            // --- Phase 1: ToolHeadLock verification ------------------------------------
            // Cmd_Extend is held TRUE for the whole of PAUSED (see the ToolHeadLock section
            // at the bottom of this FB), so the lock is already COMMANDED in the entire time
            // the machine sits paused. This phase adds the WAIT, not the command.
            //
            // Why it is needed: PAUSED used to go straight to RUNNING, so nothing re-checked
            // the lock on resume. FC_CylinderDispatch is not gated on machine state, so an
            // operator can retract the lock from the manual cylinder page while paused — in
            // cylinder FB State 3 the Cmd_Retract/Cmd_RetractFull test comes BEFORE the
            // process's Cmd_Extend, so the HMI button wins. It also catches a purely
            // mechanical failure to re-engage, which no HMI-side gate would ever see.
            //
            // Same three-way test and same error code as STATE_LOCK_EXTEND_WAIT (17), so the
            // two lock-confirm paths cannot drift apart. It cannot hang: Cmd_Extend is
            // asserted throughout, so the cylinder FB reaches either AtSetpoint or its own
            // Timeout_Extend → Error. Error_Text/ErrorDetail name the resume path so the
            // online trail still distinguishes this from a state-17 failure.
            IF #bResumeLockChk THEN
                IF "DB_HMI".Bypass_ToolHeadLock OR "DB_Cylinder_ToolHeadLock".AtSetpoint THEN
                    #bResumeLockChk := FALSE;
                    #bResumeSpeedup := TRUE;      // lock confirmed → start the spindle spin-up
                ELSIF "DB_Cylinder_ToolHeadLock".Error THEN
                    #bResumeLockChk := FALSE;
                    #newErrorFlag := TRUE;
                    #newErrorCode := 16#0012;
                    "DB_Diagnostic".Error_Text := 'PauseResume: ToolHeadLock not engaged - CylFB.Error=TRUE, AtSetpoint=FALSE';
                    "DB_HMI".ErrorDetail    := 'Tool head lock not engaged on resume - check cylinder/sensor';
                    #State := STATE_ERROR;
                END_IF;
            END_IF;

            // --- Phase 2: spindle spin-up ----------------------------------------------
            IF #bResumeSpeedup AND #tonResumeSpeedup.Q THEN
                #bResumeSpeedup := FALSE;
                #bPauseActive   := FALSE;
                #State          := STATE_RUNNING;
            END_IF;

        // -----------------------------------------------------------------
        // === STATE_TOOL_CHANGE (30) ===
        // -----------------------------------------------------------------
        30: // TOOL_CHANGE
            #StatusID := 4; #bToolExecute := TRUE; #State := STATE_TOOL_WAIT;

        // -----------------------------------------------------------------
        // === STATE_TOOL_WAIT (35) ===
        // -----------------------------------------------------------------
        35: // TOOL_WAIT
            IF #fbToolChanger.Done THEN
                #bToolExecute := FALSE;
                #CurrentTool := #fbToolChanger.CurrentTool;
                #fbRecipeHandler.ToolChangeReq := FALSE;  // Signal RecipeHandler to continue
                // Tool change done: re-engage lock before resuming machining
                #State := STATE_LOCK_EXTEND_WAIT;
            ELSIF #fbToolChanger.Error THEN
                #bToolExecute := FALSE;
                #State := STATE_ERROR;
                #newErrorFlag := TRUE;
                #newErrorCode := #fbToolChanger.ErrorID;
                "DB_HMI".ErrorDetail    := CONCAT(IN1 := 'Tool ', IN2 := INT_TO_STRING(#activeToolReq));
            END_IF;

        // -----------------------------------------------------------------
        // === STATE_ERROR (999) ===
        // -----------------------------------------------------------------
        999: // ERROR
            #StatusID := 99; #bStartSeq := FALSE; #Error := TRUE;
            #bRecipeLoadExec := FALSE;   // a recipe copy must not stay in flight across an error ack
            #timerRunning := FALSE;  // Stop cycle timer
            #bResumeSpeedup := FALSE;  // Cancel any pending pause spin-up wait (e.g. fault during spin-up)
            #bResumeLockChk := FALSE;  // Cancel any pending pause lock verification
            // Cancel any pending STOPPING spindle-decel wait. Added with ITEM-56c, but it also
            // closes a route that already existed: STATE_STOPPING could be left for STATE_ERROR by
            // an E-Stop or safety fault, and NOTHING cleared this flag on that path (only phase 2
            // itself and the hard reset did). A stale TRUE makes the NEXT stop skip phase 1
            // entirely -- no spindle stop command, no park move, no sheet-holder release -- and
            // drop straight into phase 2 on a leftover spindleStopPT. Level-cleared here every
            // scan while faulted, so no acknowledge path can miss it.
            #bWaitingSpindleStop := FALSE;
            // Cancel the end-of-program sanding dwell (2026-08-29) and drop the spindle
            // command it raised. A safety fault (E-Stop, air) during the dwell forces
            // STATE_ERROR from COMPLETE via the safety block above, and bDrivesEnable
            // already stops the spindle -- but STATE_COMPLETE is the only block that
            // clears #bSpindleStart on this path, and it no longer runs once State is 999.
            // Level-cleared every scan while faulted, so no acknowledge path can miss it.
            #bSandActive   := FALSE;
            #bSpindleStart := FALSE;
            // Clear the BackSupport atmosphere valve — de-energises on error.
            // Cmd_Retract is deliberately NOT touched here: the end-of-recipe retract
            // block (bottom of this FB) owns it and needs it held for the retract window.
            "DB_Cylinder_BackSupport".SolAtmo_Cmd := FALSE;
            // Clear BackSupport extend (recipe CMD=40 or manual button/MDI) while faulted
            "DB_Cylinder_BackSupport".Cmd_Extend  := FALSE;
            #bMDI_Cmd40Extend                     := FALSE;
            // CMD=41 edge memory: seed with the live button state while faulted, so a
            // button held through the fault cannot fire a one-shot after acknowledge.
            #prevBtnCmd41Release := "DB_Manual".Btn_Cmd41_Release;
            #prevBtnCmd41AtmoOff := "DB_Manual".Btn_Cmd41_AtmoOff;
            #prevBtnCmd41AtmoOn  := "DB_Manual".Btn_Cmd41_AtmoOn;
            // SheetHolder Cmd_Extend is driven FALSE here by its single writer at the bottom of
            // this FB (State <> SHEET_WAIT), so it cannot hold through an error acknowledge.

            // Save current position for warm restart
            IF #savedLineIndex < 0 THEN
                #savedLineIndex := #fbRecipeHandler.CurrentLine;
                #savedProgram := #activeProgram;
            END_IF;
            "DB_HMI".ResumeLine := #savedLineIndex;   // HMI shows which line will be resumed on next Start

            // Debug: populate DB_Diagnostic with error context for easier troubleshooting
            // Error_ProcessState is deliberately NOT written here: this block only runs in
            // STATE_ERROR, so it could only ever record 999. It is captured at alarm time
            // instead -- see the guarded write before the FB_AlarmManager call.
            "DB_Diagnostic".Error_Code := #fbAlarmManager.ActiveErrorCode; // primary error source
            // If recipe handler provided an error line, prefer that
            IF "DB_Diagnostic".Recipe_CurrentLine >= 0 THEN
                "DB_Diagnostic".Error_Line := "DB_Diagnostic".Recipe_CurrentLine;
            END_IF;

            // BUG FIX: Previous implementation transitioned ackEdge → STATE_PAUSED,
            // but the recipe handler remained in its internal STATE_ERROR (999).
            // In PAUSED → Continue → STATE_RUNNING the recipe handler was not running (error state).
            // Fix: All recovery paths go to STATE_STOPPED + recipe handler is reset.
            // When operator presses Start, PRE_SCAN → STARTING → RUNNING flow starts clean.
            // ACK, Continue and Restart are blocked while E-Stop is active.
            // E-Stop must be physically released before any error acknowledgement is accepted.
            IF #ackEdge AND (#EStop_OK OR "DB_HMI".Bypass_EStop) THEN
                // Acknowledge: clear error → STOPPED. savedLineIndex kept for warm restart on next Start.
                #Error := FALSE;
                #bPauseActive := FALSE;
                #bResetRecipe := TRUE;   // Reset recipe handler to IDLE (cannot continue from state 999)
                #prevSafetyError := FALSE;   // Clear safety latch -- fresh evaluation on restart
                #bSheetWaitPhase2         := FALSE;
                #bSheetWaitPhase3         := FALSE;
                IF NOT "DB_MachineConfig".Bypass_MandrelLock THEN
                    #bMandrelRetractPending := TRUE;  // ITEM-32: deferred — spindle may still be spinning; wait SpindleStopSafeTime
                END_IF;
                #bSheetHolderRetractHold  := TRUE;  // Release sheet holder (may be extended from last run)
                #fbAlarmManager(NewError := FALSE, NewErrorCode := 0,
                                AcknowledgeError := TRUE);
                #State := STATE_STOPPED;
            ELSIF #continueEdge AND (#EStop_OK OR "DB_HMI".Bypass_EStop) THEN
                // Continue: resume from savedLineIndex on next Start (warm restart)
                #Error := FALSE;
                #bPauseActive := FALSE;
                #bResetRecipe := TRUE;
                #bSheetWaitPhase2         := FALSE;
                #bSheetWaitPhase3         := FALSE;
                IF NOT "DB_MachineConfig".Bypass_MandrelLock THEN
                    #bMandrelRetractPending := TRUE;  // ITEM-32: deferred — spindle may still be spinning; wait SpindleStopSafeTime
                END_IF;
                #bSheetHolderRetractHold  := TRUE;  // Release sheet holder
                #fbAlarmManager(NewError := FALSE, NewErrorCode := 0,
                                AcknowledgeError := TRUE);
                #State := STATE_STOPPED;
            ELSIF #restartEdge AND (#EStop_OK OR "DB_HMI".Bypass_EStop) THEN
                // Restart: explicit restart from line 0 -- clear saved position
                #Error := FALSE;
                #bPauseActive := FALSE;
                #bResetRecipe := TRUE;
                #savedLineIndex := -1;
                #savedProgram := -1;
                "DB_HMI".ResumeLine := -1;
                #bSheetWaitPhase2         := FALSE;
                #bSheetWaitPhase3         := FALSE;
                IF NOT "DB_MachineConfig".Bypass_MandrelLock THEN
                    #bMandrelRetractPending := TRUE;  // ITEM-32: deferred — spindle may still be spinning; wait SpindleStopSafeTime
                END_IF;
                #bSheetHolderRetractHold  := TRUE;  // Release sheet holder
                #fbAlarmManager(NewError := FALSE, NewErrorCode := 0,
                                AcknowledgeError := TRUE);
                #State := STATE_STOPPED;
            END_IF;
    END_CASE;

    // -----------------------------------------------------------------
    // === STATE_COMPLETE (100) ===
    // (handled as IF block outside CASE -- no new constant needed)
    // -----------------------------------------------------------------
    IF #State = 100 THEN
        #StatusID := 100; #bStartSeq := FALSE;
        #Running := FALSE;
        // Clear bSpindleStart: RUNNING no longer runs to clear it, so SpindleReqStart=TRUE
        // from the last CMD_SPINDLE_ON would keep Start=TRUE through PRE_SCAN and STARTING.
        // prevStart is reset inside FB_SpindleControl on halt Done, so the next CMD_SPINDLE_ON
        // in the new recipe generates a clean startEdge.
        // bSpindleStop is intentionally NOT cleared here. (The old comment claimed the Done
        // handler in CASE 20 sets it, and that clearing it in the same scan would cancel the
        // stop. That was already wrong before this change and is corrected 2026-08-29:
        // #bSpindleStop is set in exactly ONE place, STATE_STOPPING phase 1 -- the completion
        // path never raises it. It is cleared in STATE_STOPPED. Nothing to do here either way.)
        //
        // SANDING DWELL (2026-08-29): the one exception to "bSpindleStart is FALSE in
        // COMPLETE". While #bSandActive the spindle is deliberately re-started at
        // DB_MachineConfig.SandSpeed so the operator can sand the part before taking it off.
        // Armed once at the RUNNING -> COMPLETE transition; see the note there.
        //
        // The restart is real, not a hold-over: the recipe's final CMD=21 has already run
        // FB_RecipeHandler STATE_SPINDLE_STOP_WAIT(58) to completion, which blocks until
        // DB_Spindle.IsRunning = FALSE. So FB_SpindleControl is idle and prevStart is
        // clear -- raising bSpindleStart here produces a genuine start edge.
        //
        // #bSpindleDecelWait gates the restart: the last CMD=21 set it, and tonSpindleDecel
        // (SpindleDecelTime, T#2S) clears it. Commanding RunCmd TRUE again inside that
        // window is exactly what SpindleDecelTime exists to prevent. Costs ~2 s once.
        IF #bSandActive THEN
            IF #tonSandDwell.Q THEN
                // Dwell finished -- stop the spindle and fall back to normal COMPLETE.
                #bSandActive   := FALSE;
                #bSpindleStart := FALSE;
            ELSIF NOT #bSpindleDecelWait THEN
                "DB_Spindle".Cmd_SetSpeed := #sandSpeedClamped;
                #bSpindleStart            := TRUE;
            END_IF;
        ELSE
            #bSpindleStart := FALSE;
        END_IF;
        IF NOT "DB_MachineConfig".Bypass_MandrelLock THEN
            "DB_Cylinder_MandrelLock".Cmd_Extend := FALSE;
            #bMandrelRetractPending := TRUE;    // ITEM-32: deferred — spindle still decelerating at program end; wait SpindleStopSafeTime
        END_IF;
        // De-energise the atmosphere valve. Cmd_Retract is left alone -- the
        // end-of-recipe retract block at the bottom of this FB owns it.
        "DB_Cylinder_BackSupport".SolAtmo_Cmd := FALSE;
        // Status text. The sanding variant is deliberately explicit that the spindle is
        // TURNING -- 'Program Complete' on a screen above a spinning part is how somebody
        // reaches in. English only (ITEM-55); the Spanish comes from a WinCC text list, and
        // its key for this one is DB_HMI.SandActive, NOT MachineState -- MachineState is 100
        // for both halves of COMPLETE and cannot tell them apart. Keep the wording in step
        // with the two 'sanding' rows in tools/hmi_texts.csv.
        IF #bSandActive THEN
            "DB_HMI".StatusMsg := 'Sanding - SPINDLE TURNING';
        ELSE
            "DB_HMI".StatusMsg := 'Program Complete';
        END_IF;
        // Single-writer: ErrorText is owned by FB_AlarmManager. Completion is a status,
        // not an error -- StatusMsg above already announces it ('Done!' write removed).
        // DB_HMI.CycleCount and its #bCycleCountDone one-shot were DELETED 2026-08-15.
        // The counter was a duplicate of "DB_Production".TotalOK, and a broken one: the
        // one-shot was cleared ONLY by the hard reset, and the normal cycle
        // (COMPLETE -> Start -> RECIPE_LOAD -> ... -> COMPLETE) never passes through it,
        // so CycleCount incremented once and then stayed put until somebody pressed
        // Reset. The HMI now reads DB_Production directly -- Started / OK / NOK /
        // Stopped / Aborted, which reconcile. Do not reintroduce a second parts counter
        // in DB_HMI: two sources of truth for "how many parts" is what produced the bug.
        // ITEM-56h (2026-08-16): the `ELSIF #fbInputs.Cmd_Reset` branch that used to sit here was
        // DEAD CODE and is deleted. Cmd_Reset raises #bDoHardReset in the pre-CASE handler, which
        // sets #State := STATE_STOPPED before this IF is evaluated -- so `#State = 100` was always
        // already FALSE by the time a Reset could have been seen here. It claimed that Reset from
        // COMPLETE re-loads and re-scans the recipe; it never did, and Reset from COMPLETE has
        // always meant the same as Reset anywhere else: go to STOPPED. User confirmed 2026-08-16
        // that no other meaning is wanted. Start / Restart below are the live re-run path.
        IF #fbInputs.Cmd_Start OR #restartEdge THEN
            #bResetRecipe := TRUE;      // Reset FB_RecipeHandler (state 99→0) before re-run
            // Start cancels the sanding dwell (2026-08-29). The first two lines are required:
            // nothing between here and STATE_RUNNING clears bSpindleStart, so leaving it
            // TRUE would carry the sanding speed into RECIPE_LOAD / PRE_SCAN / STARTING and
            // spin the mandrel while the operator loads the next sheet in SHEET_WAIT.
            //
            // bSpindleDecelWait is armed only if the dwell was actually turning the spindle.
            // Dropping RunCmd and then letting the new recipe's first CMD=20 raise it again is
            // precisely the case SpindleDecelTime guards, and this is the one path that can
            // reach a CMD=20 quickly after a stop the recipe handler did not issue. In practice
            // SHEET_WAIT's two-button confirm makes it much longer than T#2S, so this is cheap
            // insurance rather than an observed fault -- the flag self-clears via tonSpindleDecel
            // and, with bSpindlePendingStart FALSE, expiry does nothing else.
            IF #bSandActive THEN
                #bSpindleDecelWait := TRUE;
            END_IF;
            #bSandActive   := FALSE;
            #bSpindleStart := FALSE;
            #State := STATE_RECIPE_LOAD; // Restart/Start = immediate re-run, keeps drives on
        END_IF;
    END_IF;

    // =========================================================================
    // REFERENCE-VALIDITY LATCH (bRequireHoming)
    // =========================================================================
    // Forces a full homing cycle on the next auto start after anything that can
    // invalidate the axis reference. This is the ONLY guarantee that an E-Stop is
    // always followed by a re-home: DB_MachineConfig.AlwaysHomeOnAutoStart is an
    // operator convenience switch and must never be able to suppress this.
    //
    // Why not rely on Axis_*.StatusBits.HomingDone alone: whether the TO clears it
    // when MC_Power drops is encoder-type dependent, and an open-loop axis can lose
    // steps while the drive is dead yet still report HomingDone=TRUE on power-up.
    //
    // Placed AFTER the state machine so a STATE_ERROR transition made earlier in this
    // same scan is caught immediately rather than one scan late.
    // Cleared ONLY where a homing sequence actually completes (STATE_HOMING, both the
    // tool-axis and Bypass_ToolAxis exits). Power-up sets it TRUE (bInitDone block); a reset
    // sets it only when pressed from a state where an axis could have been moving.
    IF NOT (#EStop_OK OR "DB_HMI".Bypass_EStop) OR #State = STATE_ERROR THEN
        #bRequireHoming := TRUE;
    END_IF;

    // Drive power removed = reference lost. Level-triggered, so the latch stays TRUE for as
    // long as the drives are down and is only released by a completed homing cycle afterwards.
    //
    // This is the honest detector for the case StatusBits.HomingDone cannot see: these motors
    // are open-loop, so with the contactor open the axis can be pushed by hand or back-driven
    // by gravity while the TO happily keeps reporting the last commanded position. It is also
    // what makes it safe for a Reset pressed in MANUAL to skip homing -- if the operator turned
    // drive power off to move something by hand, this catches it regardless of the state.
    //
    // Tool axis added 2026-08-16, once Btn_Enable_Tool existed to pair with the contactor.
    // The gap it closes: Btn_Contactor_Tool is an operator toggle on the MANUAL > MANAGE screen,
    // so the tool contactor can be switched off on its own while X and Z stay powered. The
    // turret is then de-energised and can be turned by hand, and because the axis is open-loop
    // StatusBits.HomingDone stays TRUE -- so bRefTrusted is satisfied and the next start
    // presents the wrong tool angle. Exactly the case this latch exists for.
    //
    // The Bypass_ToolAxis term is mandatory, not decorative: with the bypass set,
    // Btn_Contactor_Tool is FALSE by design, so without it the latch would be permanently TRUE
    // and a bypassed machine would home on every single start. That was the original reason the
    // tool axis was left out entirely; one condition solves it.
    //
    // In auto this term cannot fire on its own -- STATE_STARTING sets all three contactor/enable
    // pairs in the same scan and only E-Stop drops them, which drops X and Z too. It earns its
    // place on the MANUAL path.
    //
    // Power-up consequence (intended): DB_HMI is NON_RETAIN, so these are FALSE until the first
    // STATE_STARTING asserts them -- the latch is held TRUE until the machine has been started
    // once and homed, which is exactly the required power-up behaviour.
    IF NOT ("DB_HMI".Btn_Contactor_X AND "DB_HMI".Btn_Enable_X)
       OR NOT ("DB_HMI".Btn_Contactor_Z AND "DB_HMI".Btn_Enable_Z)
       OR (NOT "DB_MachineConfig".Bypass_ToolAxis
           AND NOT ("DB_HMI".Btn_Contactor_Tool AND "DB_HMI".Btn_Enable_Tool)) THEN
        #bRequireHoming := TRUE;
    END_IF;

    "DB_Diagnostic".Require_Homing := #bRequireHoming;  // HMI/diagnostic visibility

    // =========================================================================
    // CYCLE TIMER - runs during RUNNING and PAUSED
    // =========================================================================
    #tonElapsed(IN := #timerRunning, PT := T#24h);
    // Homing timeout: counts only while in STATE_HOMING; auto-resets when state exits
    #tonHomingTimeout(IN := (#State = STATE_HOMING), PT := "DB_MachineConfig".Timeout_Homing);
    // ITEM-30: independent timeout for STATE_STOP_GOHOME — gets a full budget regardless of
    // how much time was consumed by the preceding STATE_HOMING sequence earlier in the same run
    #tonStopHomeTimeout(IN := (#State = STATE_STOP_GOHOME), PT := "DB_MachineConfig".Timeout_Homing);
    // ToolHeadLock wait: counts in both lock wait states; auto-resets on exit
    // tonLockWait: 3s total (1s pre-delay + up to 2s for cylinder stroke). AtSetpoint exits early.
    #tonLockWait(IN := (#State = STATE_LOCK_RETRACT_WAIT),
                 PT := "DB_MachineConfig".CylToolHeadLock_RetractTime);
    #tonLockPreDelay(IN := (#State = STATE_LOCK_EXTEND_WAIT), PT := "DB_MachineConfig".CylToolHeadLock_PreDelay);
    // Spindle-stop wait: safety fallback for MandrelLock retract in STATE_STOPPING.
    // Duration = (capturedSpindleRPM / SpindleMaxRPM) * SpindleStopSafeTime. Fires immediately if speed was 0.
    #tonSpindleStopWait(IN := (#State = STATE_STOPPING AND #bWaitingSpindleStop), PT := #spindleStopPT);
    // MandrelLock stroke wait: open-loop during STATE_SHEET_WAIT phase 2
    #tonMandrelWait(IN := (#State = STATE_SHEET_WAIT AND #bSheetWaitPhase2), PT := "DB_MachineConfig".CylMandrelLock_ClampTime);
    // SheetHolder retract wait: open-loop during STATE_SHEET_WAIT phase 3
    #tonSheetHolderRetract(IN := (#State = STATE_SHEET_WAIT AND #bSheetWaitPhase3), PT := "DB_MachineConfig".CylSheetHolder_RetractTime);
    // ITEM-32: safety gate timer for deferred MandrelLock retract.
    // Six unsafe paths (Reset/Error-ack/Error-restart/Error-continue/Restart-pre-CASE/Complete) set
    // bMandrelRetractPending instead of bMandrelRetractPulse. This timer counts SpindleStopSafeTime
    // to ensure the spindle has physically stopped before the mandrel lock releases.
    // bMandrelRetractPending is NOT cleared by bDoHardReset — it must stay TRUE until the timer fires.
    #tonMandrelRetractWait(IN := #bMandrelRetractPending, PT := "DB_MachineConfig".SpindleStopSafeTime);
    // MandrelLock one-shot retract pulse (still ValveType=1, 5/2 spring return):
    // ValveType=1 + Mode=0 keeps Sol_A=TRUE in State 3 even after Cmd_Extend=FALSE.
    // A one-scan Cmd_Retract=TRUE pulse forces the FB to State 2 (Sol_A=FALSE) → spring retracts.
    // ITEM-32: promote deferred retract to immediate pulse once safety timer has elapsed.
    // STATE_STOPPING uses bMandrelRetractPulse directly (already waited proportional timer) — no change there.
    IF #tonMandrelRetractWait.Q THEN
        #bMandrelRetractPulse   := TRUE;   // Fire the retract this scan
        #bMandrelRetractPending := FALSE;  // Clear pending; timer IN drops next scan → ET resets
    END_IF;
    "DB_Cylinder_MandrelLock".Cmd_Retract  := #bMandrelRetractPulse;
    #bMandrelRetractPulse := FALSE;  // Self-clearing: active for exactly one scan

    // =========================================================================
    // SHEETHOLDER COMMANDS -- single writer for BOTH directions (ITEM-46)
    // =========================================================================
    // ValveType=2, 5/3 blocked centre, PositioningMode=0. There is no spring on this
    // cylinder any more, so:
    //   Cmd_Extend  = TRUE only while the sheet must be held: STATE_SHEET_WAIT Ph1
    //                 (operator inserting) and Ph2 (MandrelLock clamping). FALSE in
    //                 every other state, on every path, without exception.
    //   Cmd_Retract = HELD for the retract stroke, then dropped -> both coils off and
    //                 the blocked centre holds the piston at the retract end.
    //
    // Why Cmd_Extend is written here instead of inside the states (fixes the "retracts,
    // then extends again a second later" stop bug): STATE_SHEET_WAIT Ph1 used to latch
    // Cmd_Extend and only STOPPED / ERROR cleared it. Pressing Stop during Ph1/Ph2 goes
    // to STOPPING (18) -> LOCK_RETRACT_WAIT (29) -> STOPPED, so Cmd_Extend stayed TRUE
    // for several seconds while Cmd_Retract was also held. The cylinder FB retracted,
    // hit Timeout_Retract, landed in State 4, saw Cmd_Extend still TRUE and extended
    // straight back out. Driving Cmd_Extend from the state itself makes that impossible.
    //
    // Why the retract is time-bounded instead of released on FB State 4: in Mode 0 with a
    // 5/3 valve, State 4 keeps Sol_B energised for ever (09_Sensors_Actuators.scl State-4
    // output branch) and is left only on a new extend command -- so the coil stayed live
    // the whole time the machine sat idle, from the first power-up retract onwards. With
    // Timeout_Retract = T#24H the FB now stays in State 2 for the whole hold, and dropping
    // the latch takes it to State 0 (09: "NOT Cmd_Retract") -> both coils off.
    //
    // Deterministic clear path (Reset-Path Rule checkpoints 1-4):
    //   - The TON below always ends the hold, in EVERY state. It is deliberately not a
    //     state test: STOPPED / ERROR are reached mid-retract and the latch commands the
    //     SAFE direction there, so it must be the timer that ends it, never the state.
    //   - Cleared again in STATE_SHEET_WAIT Ph1 before an extend is commanded.
    //   - The timer needs no explicit IN := FALSE: IN is the latch itself, so every path
    //     that clears or re-arms the latch resets ET with it.
    "DB_Cylinder_SheetHolder".Cmd_Extend :=
        (#State = STATE_SHEET_WAIT) AND NOT #bSheetWaitPhase3;

    // Cmd_Release: drop the coil hold WITHOUT moving the piston (5/3 blocked centre).
    //
    // The extend side has the same dead end ITEM-46 fixed on the retract side: with
    // PositioningMode=0 the cylinder FB latches Sol_A ON in State 3 (AT SETPOINT) and the only
    // exits are a new extend or a retract command. The holder reaches State 3 after
    // Timeout_Extend during SHEET_WAIT Ph1 -- correct while the operator is loading, since the
    // blank is being held -- but if the machine faults there, dropping Cmd_Extend is not enough:
    // Sol_A stays energised for however long the machine sits in ERROR waiting for an Ack.
    //
    // Releasing is NOT the same as retracting, and that distinction is the whole point. A retract
    // would let go of a blank that MandrelLock has not clamped yet (a fault in Ph1/Ph2 is exactly
    // when that is true, and it is the only time the holder is extended at all). Cmd_Release takes
    // the FB to State 0 instead: both coils off, and the blocked centre holds the piston exactly
    // where it is. Same physical outcome the machine already accepts on E-Stop, where
    // FB_CylinderControl forces State -1 and de-energises everything.
    //
    // Asserted in ERROR and STOPPED (Reset-Path Rule checkpoints 3 and 4: no actuator override may
    // stay latched in either). In STOPPED it is a no-op on every traced path -- every route to
    // STOPPED runs a retract first, which ends in State 0 anyway -- but it is the deterministic
    // guard if a future path ever leaves the FB holding while the machine is idle.
    // The operator's Ack still performs the actual release: it arms bSheetHolderRetractHold, and
    // State 0 accepts Cmd_Retract normally.
    "DB_Cylinder_SheetHolder".Cmd_Release :=
        (#State = STATE_ERROR) OR (#State = STATE_STOPPED);

    #tonSheetHolderHold(IN := #bSheetHolderRetractHold AND (#EStop_OK OR "DB_HMI".Bypass_EStop),
                        PT := "DB_MachineConfig".CylSheetHolder_RetractTime);
    IF #tonSheetHolderHold.Q THEN
        #bSheetHolderRetractHold := FALSE;
    END_IF;
    "DB_Cylinder_SheetHolder".Cmd_Retract  := #bSheetHolderRetractHold;
    // Drive ready timeout: counts while in STARTING and drives not yet ready; auto-resets on exit.
    // Same tool term as the STARTING readiness test above -- the two must agree, or the state
    // waits on a condition the timeout is not counting against (or vice versa).
    #tonDriveReady(IN := (#State = STATE_STARTING)
                         AND NOT (#fbPowerX.Status AND #fbPowerZ.Status
                                  AND (#fbPowerTool.Status OR "DB_MachineConfig".Bypass_ToolAxis)),
                   PT := "DB_MachineConfig".Timeout_DriveReady);
    // Spindle decel wait: blocks RunCmd from going TRUE until VFD ramp-down completes
    #tonSpindleDecel(IN := #bSpindleDecelWait, PT := "DB_MachineConfig".SpindleDecelTime);
    // Pause resume spin-up wait: counts while bResumeSpeedup (Continue pressed in PAUSED).
    // IN drops to FALSE on reset/stop/error via bResumeSpeedup clears → ET resets, no stale fire.
    #tonResumeSpeedup(IN := #bResumeSpeedup, PT := "DB_MachineConfig".SpindleResumeSpeedupTime);
    // End-of-program sanding dwell (2026-08-29). IN is gated on #bSpindleStart, not on
    // #bSandActive alone, so the clock only runs while the spindle is actually commanded --
    // the operator gets the full SandTime_s of turning part, not SandTime_s minus the
    // SpindleDecelTime window that STATE_COMPLETE waits out before restarting.
    // Also gated on E-Stop, same as tonSheetHolderHold: an E-Stop mid-dwell pauses the
    // timer rather than burning it with the drive dead. (The safety block normally forces
    // STATE_ERROR first, which clears #bSandActive outright; this is the belt-and-braces
    // case where the E-Stop is bypassed but the drive is down for another reason.)
    // PT comes from #sandTimePT (clamped seconds -> Time, computed before the CASE), never
    // straight from the config -- SandTime_s is an Int of seconds, not a Time.
    #tonSandDwell(IN := #bSandActive AND #bSpindleStart
                        AND (#EStop_OK OR "DB_HMI".Bypass_EStop),
                  PT := #sandTimePT);
    IF #tonSpindleDecel.Q THEN
        #bSpindleDecelWait := FALSE;
        IF #bSpindlePendingStart THEN
            "DB_Spindle".Cmd_SetSpeed := #pendingSpindleSpeed;
            #bSpindleStart        := TRUE;
            #bSpindlePendingStart := FALSE;
        END_IF;
    END_IF;
    IF #timerRunning THEN
        "DB_HMI".ElapsedTime := #tonElapsed.ET;
        "DB_HMI".ElapsedSeconds := TIME_TO_DINT(#tonElapsed.ET / 1000);
    END_IF;
    // Reset timer on new program start
    IF #State = STATE_STARTING THEN
        #tonElapsed(IN := FALSE, PT := T#24h);  // Reset
        "DB_HMI".ElapsedTime := T#0s;
        "DB_HMI".ElapsedSeconds := 0;
    END_IF;

    // =========================================================================
    // PRODUCTION LOGGING - DB_Production
    // =========================================================================
    // Edge: cycle start (enter RECIPE_LOAD).
    //
    // This was the PRE_SCAN(12) edge until 2026-08-15. RECIPE_LOAD(11) runs one state
    // EARLIER, and it is the first state every accepted Start press reaches -- from
    // STOPPED, from MANUAL and from COMPLETE alike. Counting at PRE_SCAN meant a start
    // that died in the recipe copy (16#0312 transfer refused, 16#0314 chunk never
    // arrived, 16#0316 checksum mismatch) incremented nothing: TotalStarted had not
    // fired yet, and CurrentActive was still FALSE so the STATE_ERROR edge below
    // skipped it too. Those failures were invisible to the production counters --
    // exactly the ones worth counting while the chunked transfer is still on trial.
    //
    // Counting here also makes CurrentStartTime the time of the Start press rather than
    // the time the copy finished, and it is what makes the TotalStarted invariant in
    // DB_Production hold: every accepted start now has an outcome bucket waiting for it.
    //
    // Safe as a single edge: RECIPE_LOAD is never re-entered from within a cycle (it
    // exits to PRE_SCAN on Done or to ERROR on failure, and nothing loops back), so this
    // fires exactly once per Start.
    IF (#State = STATE_RECIPE_LOAD) AND (#prevState <> STATE_RECIPE_LOAD) THEN
        "DB_Production".CurrentActive := TRUE;
        "DB_Production".CurrentProgram := #activeProgram;
        "DB_Production".TotalStarted := "DB_Production".TotalStarted + 1;
        #prodTimeStatus := RD_SYS_T(OUT => #prodTimeNow);
        "DB_Production".CurrentStartTime := #prodTimeNow;
    END_IF;

    // Edge: OK complete (enter state 100)
    IF (#State = 100) AND (#prevState <> 100) THEN
        "DB_Production".LastResult := 1;  // OK
        "DB_Production".LastProgram := #activeProgram;
        "DB_Production".LastDuration_s := "DB_HMI".ElapsedSeconds;
        "DB_Production".LastErrorCode := 0;
        "DB_Production".LastErrorLine := -1;
        "DB_Production".TotalOK := "DB_Production".TotalOK + 1;
        #prodTimeStatus := RD_SYS_T(OUT => #prodTimeNow);
        "DB_Production".LastEndTime := #prodTimeNow;
        "DB_Production".CurrentActive := FALSE;
        // History ring push removed 2026-07-31 (memory reclaim) -- see DB_Production
        // in 02_DataBlocks.scl. Last* summary above is the surviving record.
    END_IF;

    // Edge: NOK (enter STATE_ERROR with active cycle)
    IF (#State = STATE_ERROR) AND (#prevState <> STATE_ERROR) AND "DB_Production".CurrentActive THEN
        "DB_Production".LastResult := 2;  // NOK
        "DB_Production".LastProgram := #activeProgram;
        "DB_Production".LastDuration_s := "DB_HMI".ElapsedSeconds;
        "DB_Production".LastErrorCode := #fbAlarmManager.ActiveErrorCode;
        "DB_Production".LastErrorLine := "DB_Diagnostic".Error_Line;
        "DB_Production".TotalNOK := "DB_Production".TotalNOK + 1;
        #prodTimeStatus := RD_SYS_T(OUT => #prodTimeNow);
        "DB_Production".LastEndTime := #prodTimeNow;
        "DB_Production".CurrentActive := FALSE;
        // History ring push removed 2026-07-31 (memory reclaim) -- see DB_Production
        // in 02_DataBlocks.scl. Fault detail is retained in DB_AlarmHistory / DB_Error.
    END_IF;

    // Edge: cycle ended at STOPPED with a cycle still in flight.
    //
    // Trigger is ANY entry to STOPPED (#prevState <> STOPPED) with CurrentActive set --
    // not a whitelist of "expected" previous states. It used to be a whitelist of
    // {STOPPING, STOP_GOHOME, STOP_GOTOZERO, LOCK_RETRACT_WAIT}, which counted an
    // operator STOP correctly and lost everything else: bDoHardReset sets
    // State := STOPPED DIRECTLY from RUNNING / PAUSED / SHEET_WAIT / HOMING / whatever,
    // so a Reset pressed mid-cycle hit no bucket at all, and left CurrentActive stranded
    // TRUE until the next start happened to overwrite it. TotalStarted then permanently
    // exceeded the sum of the outcomes with no record of where the difference went.
    //
    // A whitelist here fails OPEN -- a state added later that reaches STOPPED by a new
    // route silently stops being counted. Counting every entry and then classifying it
    // fails CLOSED: an unrecognised route lands in TotalAborted, which is visible and
    // wrong-looking rather than invisible.
    //
    // No double-count risk: the two other terminal edges (COMPLETE and ERROR, above)
    // both clear CurrentActive on the scan they fire, so the STOPPED that follows an
    // error acknowledge or a stop-from-COMPLETE finds it already FALSE.
    IF (#State = STATE_STOPPED) AND (#prevState <> STATE_STOPPED)
       AND "DB_Production".CurrentActive THEN
        "DB_Production".LastProgram := #activeProgram;
        "DB_Production".LastDuration_s := "DB_HMI".ElapsedSeconds;
        "DB_Production".LastErrorCode := 0;
        "DB_Production".LastErrorLine := -1;
        #prodTimeStatus := RD_SYS_T(OUT => #prodTimeNow);
        "DB_Production".LastEndTime := #prodTimeNow;
        "DB_Production".CurrentActive := FALSE;
        IF (#prevState = STATE_STOPPING) OR (#prevState = STATE_LOCK_RETRACT_WAIT)
           OR (#prevState = STATE_STOP_GOHOME) OR (#prevState = STATE_STOP_GOTOZERO) THEN
            // Operator pressed Stop: the machine ran its park sequence and the axes
            // finished at the sheet-load position. A clean, planned end.
            "DB_Production".LastResult := 3;  // STOP
            "DB_Production".TotalStopped := "DB_Production".TotalStopped + 1;
        ELSE
            // Any other route to STOPPED with a cycle active -- in practice Reset
            // pressed from an active state. Deliberately NOT merged into TotalStopped:
            // a Stop parks the axes, a Reset does not, so the two say different things
            // about where the machine was left and are worth telling apart.
            "DB_Production".LastResult := 4;  // ABORT
            "DB_Production".TotalAborted := "DB_Production".TotalAborted + 1;
        END_IF;
        // History ring push removed 2026-07-31 (memory reclaim) -- see DB_Production
        // in 02_DataBlocks.scl. Last* summary above is the surviving record.
    END_IF;

    // Production RESET: clear counters (history ring removed 2026-07-31)
    IF #prodResetEdge THEN
        "DB_Production".TotalStarted := 0;
        "DB_Production".TotalOK := 0;
        "DB_Production".TotalNOK := 0;
        "DB_Production".TotalStopped := 0;
        "DB_Production".TotalAborted := 0;   // must be zeroed with the rest or the
                                             // TotalStarted invariant breaks after a reset
        // Optionally also clear last cycle summary
        "DB_Production".LastResult := 0;
        "DB_Production".LastProgram := 0;
        "DB_Production".LastDuration_s := 0;
        "DB_Production".LastErrorCode := 0;
        "DB_Production".LastErrorLine := -1;
        "DB_Production".CurrentActive := FALSE;
    END_IF;

    // Last-cycle RESET: only clear last cycle summary (counters and history are preserved)
    IF #lastCycleResetEdge THEN
        "DB_Production".LastResult := 0;
        "DB_Production".LastProgram := 0;
        "DB_Production".LastDuration_s := 0;
        "DB_Production".LastErrorCode := 0;
        "DB_Production".LastErrorLine := -1;
    END_IF;

    // Update prevState for next cycle
    #prevState := #State;

    // =========================================================================
    // RECIPE HANDLER + PRE-SCAN - Execute based on active program
    // =========================================================================
    // Both FBs are called EVERY scan regardless of machine state.
    // fbPreScan: Execute=bPreScanExec is TRUE only inside STATE_PRE_SCAN; all
    // other states call it with FALSE so its internal state machine returns
    // DONE(99) -> IDLE(0) and rearms its rising-edge start for the next run.
    // (BUG FIX: previously called only inside STATE_PRE_SCAN with Execute held
    // TRUE, so validation only ever ran on the first cycle after power-up.)
    // 2026-08-04: was a five-way CASE binding DB_RecipeProgram1..5. Those DBs
    // now live in load memory and cannot be passed as an InOut reference at all.
    // Both FBs bind unconditionally to DB_SelectedRecipe, which STATE_RECIPE_LOAD(11)
    // fills before the pre-scan runs. One call site, no per-program duplication.
    // Reset wiring mirrors fbRecipeHandler below. NOTE: bDoHardReset must NOT be
    // used here -- the hard-reset block clears it earlier in this same scan, so it
    // is always FALSE by the time we get here. bResetRecipe is the one-shot with
    // the right lifecycle: set by the hard reset AND by every start path, consumed
    // here, cleared a few lines further down.
    #fbRecipeLoader(Execute   := #bRecipeLoadExec,
                    ProgramNo := #activeProgram,
                    Reset     := #fbInputs.Cmd_Reset OR #bResetRecipe);

    #fbRecipeHandler(Start := #bStartSeq, Stop := #fbInputs.Cmd_Stop,
                     Pause := #bPauseActive, Reset := #fbInputs.Cmd_Reset OR #bResetRecipe,
                     bStartEdge := #fbInputs.Cmd_Start,
                     StartLine := MAX(IN1 := INT#0, IN2 := #savedLineIndex),
                     LineCount := #activeLineCount,
                     Lines := "DB_SelectedRecipe".Lines,
                     Axis_X := #Axis_X, Axis_Z := #Axis_Z);
    #fbPreScan(Execute := #bPreScanExec, LineCount := #activeLineCount,
               Lines := "DB_SelectedRecipe".Lines);

    // bResetRecipe is a ONE-SHOT: self-cleared here, right after the handler call that
    // consumed it (same pattern as bHaltAllAxes below). Every setter runs earlier in the
    // scan (hard reset, STOPPED/MANUAL Start, ERROR ack/continue/restart, COMPLETE), so
    // the handler always sees it for exactly one scan.
    //
    // BUG FIX 2026-07-31: it used to be cleared ONLY in STATE_PRE_SCAN, so after power-up,
    // after any Cmd_Reset, and after an error acknowledge it stayed TRUE for as long as the
    // machine sat in STOPPED or MANUAL -- i.e. exactly when the operator uses the manual
    // page. FB_RecipeHandler is called every scan and its `IF #Reset THEN` block is level-
    // triggered, so it re-cleared BackSupport Cmd_Extend / Cmd_Retract / SolAtmo_Cmd every
    // scan, wiping the manual CMD=40/CMD=41 buttons and the MDI (both write earlier in the
    // scan, in the STATE_MANUAL branch). Nothing ever reached the OB1 output assignment.
    //
    // 2026-08-04: the program-number guard is gone. It existed because the old
    // five-way CASE called no handler at all outside 1..5, so the flag had to
    // survive to a scan where one ran. fbRecipeHandler is now called every scan
    // unconditionally, so it always consumes the flag immediately.
    #bResetRecipe := FALSE;

    // =========================================================================
    // END-OF-RECIPE BACKSUPPORT RETRACT  (operator spec 2026-08-07)
    // =========================================================================
    // "When a recipe is finished, fail or successful, de-energise Sol_A, Sol_B and
    //  SolAtmo -- retract with Sol_B for 2 s, then turn off -- so every next recipe
    //  can start clean."
    //
    // Deliberately placed AFTER the #fbRecipeHandler call above: the handler's
    // level-triggered `IF #Reset THEN` block also writes BackSupport commands, so
    // FB_Process must be the LAST writer of Cmd_Retract or the two would fight
    // within a single scan.
    //
    // EDGE, not level: STOPPED / ERROR / COMPLETE all run every scan while the
    // machine sits idle, so a level trigger would restart the retract forever.
    // bBSTerminalPrev is seeded TRUE by the bInitDone FIRST-SCAN block, so power-up
    // (which begins in STOPPED) does not fire an unexpected retract.
    //
    // The seed must NOT be moved into the general bDoHardReset block, however natural
    // that reads: bDoHardReset sets State := STOPPED at its top, so a pre-seeded edge
    // memory turns a Reset pressed while RUNNING into terminal->terminal -- no edge, no
    // retract, cylinder frozen mid-recipe. Nor may bDoHardReset clear bBSEndRetract: a
    // Reset landing inside the retract window would abandon the piston mid-stroke.
    // Both mistakes were made and caught on review 2026-08-09; see TODO.md ITEM-48.
    //
    // MANUAL(5) -> STOPPED(0) also fires this, because MANUAL is not a terminal
    // state. That is NOT a bug -- operator confirmed 2026-08-07 that retracting on
    // the way out of manual is wanted. A `#prevState <> STATE_MANUAL` guard was
    // offered and declined. Do not add one.
    #bBSTerminalNow := (#State = STATE_STOPPED) OR (#State = STATE_ERROR) OR (#State = 100);

    IF #bBSTerminalNow AND NOT #bBSTerminalPrev THEN
        #bBSEndRetract := TRUE;               // entered a terminal state this scan
    END_IF;
    IF NOT #bBSTerminalNow THEN
        IF #bBSEndRetract THEN
            // Left a terminal state part-way through the retract window (Start pressed, or
            // MANUAL entered). Drop Cmd_Retract together with the latch: nothing else in
            // this FB clears it, and the MANUAL route never raises bResetRecipe, so without
            // this the cylinder would be held retracting for the whole manual session.
            "DB_Cylinder_BackSupport".Cmd_Retract := FALSE;
        END_IF;
        #bBSEndRetract := FALSE;
    END_IF;
    #bBSTerminalPrev := #bBSTerminalNow;

    // Gated on E-Stop for the same reason as tonSheetHolderHold: FB_CylinderControl forces
    // State -1 and drops every coil while SafetyOK is FALSE (OB1 passes the same signal), so
    // an E-Stop during the window would run the timer out with the piston never moving and
    // leave the BackSupport frozen mid-stroke. Pausing the window instead means the retract
    // completes as soon as the E-Stop is released.
    #tonBSEndRetract(IN := #bBSEndRetract AND (#EStop_OK OR "DB_HMI".Bypass_EStop),
                     PT := "DB_MachineConfig".CylBackSupport_EndRetractTime);

    IF #bBSEndRetract THEN
        "DB_Cylinder_BackSupport".SolAtmo_Cmd := FALSE;   // atmosphere off for the whole sequence
        IF #tonBSEndRetract.Q THEN
            // Retract time elapsed: release Cmd_Retract. FB State 2 -> State 0
            // (09:617-619); Sol_A and Sol_B both drop and the 5/3 blocked centre
            // holds the piston where it stopped. This is the "all coils off" state.
            "DB_Cylinder_BackSupport".Cmd_Retract := FALSE;
            #bBSEndRetract := FALSE;
        ELSE
            // FB State 3 (or 0) -> State 2: Sol_A off, Sol_B on (09:828-830).
            // Cmd_Extend must go first -- State 1 ignores Cmd_Retract while it is held.
            "DB_Cylinder_BackSupport".Cmd_Extend  := FALSE;
            "DB_Cylinder_BackSupport".Cmd_Retract := TRUE;
        END_IF;
    END_IF;

    // Homing -- sequential pattern: STATE_HOMING (startup) and STATE_STOP_GOHOME (post-stop)
    // both use homeSeqState + bHomeXExec/bHomeZExec.
    //
    // MODE. Always 3 -- active + zero: seek the reference switch, then set the position.
    // A literal, deliberately. DB_Manual.HomingMode is NOT read here: it belongs to
    // FB_ManualMode's own MC_Home instances (see the FB_ManualMode call near the bottom
    // of this FB), and letting a manual-screen setting change the AUTOMATIC homing mode
    // is not something anyone would intend. User-confirmed 2026-09-06.
    //
    // This replaces three SEL() calls whose polarity was INVERTED against the comment
    // that described them (fixed 2026-09-06). SEL returns IN0 when G is FALSE, so
    //     SEL(G := (State = STATE_HOMING AND ...), IN0 := 3, IN1 := DB_Manual.HomingMode)
    // used DB_Manual.HomingMode *inside* STATE_HOMING and 3 everywhere else -- the exact
    // opposite of "mode 3 is forced in STATE_HOMING". It was invisible because
    // FC_LoadConfig sets DB_Manual.HomingMode := 3, so both branches evaluated to 3. It
    // would have surfaced the first time anyone changed the manual homing mode -- which
    // is exactly what that tag is FOR, so this was a live trap, not a theoretical one.
    // Do not re-couple them, and do not reintroduce a SEL here: the polarity is what
    // misled every reader of the original.
    //
    // A DB_HMI.Sim_HomeInPlace flag briefly lived here (2026-09-06) to pick Mode 0 for
    // PLCSIM. It was REVERTED the same day: S7-PLCSIM does not simulate S7-1200 motion
    // control at all -- the technology objects download but their logic does not run, and
    // the PTO hardware is not simulated -- so MC_Home never completes in ANY mode and the
    // flag could not do what it was written for. Do not re-add it. See CLAUDE.md.
    #fbHomeX(
        Execute := #bHomeXExec,
        Mode := 3,
        Position := "DB_MachineConfig".HomeOffset_X,
        Axis := #Axis_X
    );
    #fbHomeZ(
        Execute := #bHomeZExec,
        Mode := 3,
        Position := "DB_MachineConfig".HomeOffset_Z,
        Axis := #Axis_Z
    );
    #fbHomeTool(
        Execute  := #bHomeToolExec,
        Mode     := 3,
        Position := 0.0,
        Axis     := #Axis_Tool
    );
    // PNP halt FBs: Execute stays TRUE until bHaltX/Z_PNP is cleared (on return to STATE_STOPPED)
    #fbHaltX_PNP(Execute := #bHaltX_PNP, Axis := #Axis_X);
    #fbHaltZ_PNP(Execute := #bHaltZ_PNP, Axis := #Axis_Z);
    // ITEM-31: reset/startup halt — MC_Halt rising edge fires on the scan that bDoHardReset or
    // first-scan startup set bHaltAllAxes TRUE. Aborts any MC_Home command still active in the TO.
    // bHaltAllAxes is self-cleared here (after the calls) so the rising edge occurs for exactly one scan.
    // Must NOT be cleared earlier (e.g. in STATE_STOPPED CASE) — state machine runs before this section.
    #fbHaltX_Reset(Execute    := #bHaltAllAxes, Axis := #Axis_X);
    #fbHaltZ_Reset(Execute    := #bHaltAllAxes, Axis := #Axis_Z);
    #fbHaltTool_Reset(Execute := #bHaltAllAxes, Axis := #Axis_Tool);
    #bHaltAllAxes := FALSE;  // Self-clearing: active for exactly one scan

    // Tool changer -- only rotates the turret; axis positioning done by G-code
    #fbToolChanger(Execute := #bToolExecute, ToolNumber := #activeToolReq,
                   Axis_Tool := #Axis_Tool);

    // Belt-and-braces clamp for the clearance/park move target. parkTargetX/Z are already
    // clamped (computed before the state machine); this also covers the STATE_PRE_HOME_CLR
    // target, which is derived from HomeOffset + PostHome_Clearance.
    #clrTargetX  := MIN(IN1 := MAX(IN1 := #clrTargetX,
                                   IN2 := "DB_MachineConfig".SoftLimit_MinX),
                        IN2 := "DB_MachineConfig".SoftLimit_MaxX);
    #clrTargetZ  := MIN(IN1 := MAX(IN1 := #clrTargetZ,
                                   IN2 := "DB_MachineConfig".SoftLimit_MinZ),
                        IN2 := "DB_MachineConfig".SoftLimit_MaxZ);
    // Defensive: every path that sets bHomeClrX/Z also sets clrVelocity in the same scan,
    // but a zero velocity would fail MC_MoveAbsolute rather than move slowly. Never pass 0.
    IF #clrVelocity <= 0.0 THEN
        #clrVelocity := "DB_MachineConfig".RapidVelocity;
    END_IF;

    // Stop/park move -- STATE_STOPPING sends both axes to the sheet-load park position
    // (was hardcoded 0.0 before the sheet-load park change).
    #fbMoveX_Stop(Execute := #bStopMoveX, Position := #parkTargetX, Velocity := "DB_MachineConfig".RapidVelocity, Axis := #Axis_X);
    #fbMoveZ_Stop(Execute := #bStopMoveZ, Position := #parkTargetZ, Velocity := "DB_MachineConfig".RapidVelocity, Axis := #Axis_Z);
    // Clearance / park moves. Target comes from #clrTargetX/Z, set by the caller state:
    //   STATE_PRE_HOME_CLR  (13) -- HomeOffset + PostHome_Clearance (PNP escape before homing)
    //   STATE_POST_HOME_CLR (16) -- SheetLoadPos (park for sheet loading)
    #fbMoveX_HomeClr(Execute  := #bHomeClrX,
                     Position := #clrTargetX,
                     Velocity := #clrVelocity,
                     Axis     := #Axis_X);
    #fbMoveZ_HomeClr(Execute  := #bHomeClrZ,
                     Position := #clrTargetZ,
                     Velocity := #clrVelocity,
                     Axis     := #Axis_Z);

    // Manual mode - sync aliases first
    // Soft-limit jog gating (manual): once an axis is HOMED, jogging deeper past a
    // configured soft limit is blocked; jogging back toward the valid range always
    // passes (same escape pattern as PNP below -- never fault, never trap the operator).
    // Un-homed axes are NOT gated: position is meaningless before the reference seek,
    // so soft limits cannot apply. Tool axis (SelectedAxis=2) is never gated here.
    // TOOLHEADLOCK INTERLOCK (2026-08-14) -- the turret must not be driven while the
    // lock is engaged. The lock is a pin into the turret: rotating against it damages
    // the pin, the turret, or both, and nothing downstream would notice, because an
    // open-loop stepper reports a completed move whether or not the shaft turned.
    //
    // "Engaged" is ANY of:
    //   Sol_A       the PLC is commanding extend right now. Unambiguous, and it holds
    //               even on a machine whose sensor is absent or bypassed.
    //   AtSetpoint  the sensor says the pin is in (PositioningMode = 1, real switch on
    //               this cylinder). Ignored when Bypass_ToolHeadLock is set, which is
    //               how a machine with no sensor is commissioned -- otherwise a missing
    //               switch would permanently forbid tool jogging.
    //
    // NOT tested: "the cylinder has not confirmed it is retracted". That would be the
    // stricter interlock, but this cylinder has NO retract sensor -- OB1 wires only
    // Sen_AtSetpoint, and FB_CylinderControl derives AtRetract from State 4, which is
    // only entered when Sen_AtRetract is TRUE. AtRetract is therefore permanently FALSE
    // here, and testing it would forbid tool jogging forever. The residual gap is a pin
    // stuck mid-stroke with the coil off and the sensor not made: undetectable on this
    // hardware. Wire In_Cyl_ToolHeadLock_AtRetract if that case matters, then add the
    // term -- do not add it before the sensor exists.
    //
    // In MANUAL the lock should already be retracted (FB_Process only commands extend
    // in states 17/20/25 and the 5/2 valve springs back), so this normally never fires.
    // It exists for when that assumption is wrong: a stuck spool, a failed spring, a
    // fault that left the machine in MANUAL with the pin still in.
    #bToolLockEngaged :=
        "DB_Cylinder_ToolHeadLock".Sol_A
        OR (NOT "DB_HMI".Bypass_ToolHeadLock
            AND "DB_Cylinder_ToolHeadLock".AtSetpoint);

    // Only the TOOL axis is affected. X and Z are free to move with the lock engaged --
    // that is a normal machining condition, not a fault.
    #bToolAxisBlocked := #bToolLockEngaged AND "DB_Manual".SelectedAxis = 2;

    // The turret-step buttons are gated on the lock ALONE, like HomeAll: FB_ManualMode's
    // ToolStepCW/CCW branches (state 0) do not test SelectedAxis at all -- they drive
    // MC_MoveRelative on Axis_Tool whatever axis is selected. Gating them on
    // bToolAxisBlocked would leave the hole open for every selection except 2.
    // This flag exists only to raise the banner; the refusal is the NOT bToolLockEngaged
    // term on the FB inputs below.
    #bToolStepBlocked := #bToolLockEngaged
        AND ("DB_Manual".Btn_ToolStepCW OR "DB_Manual".Btn_ToolStepCCW);

    #bJogBlockPlus :=
        ("DB_Manual".SelectedAxis = 0 AND #Axis_X.StatusBits.HomingDone
         AND #Axis_X.ActualPosition >= "DB_MachineConfig".SoftLimit_MaxX) OR
        ("DB_Manual".SelectedAxis = 1 AND #Axis_Z.StatusBits.HomingDone
         AND #Axis_Z.ActualPosition >= "DB_MachineConfig".SoftLimit_MaxZ) OR
        #bToolAxisBlocked;
    #bJogBlockMinus :=
        ("DB_Manual".SelectedAxis = 0 AND #Axis_X.StatusBits.HomingDone
         AND #Axis_X.ActualPosition <= "DB_MachineConfig".SoftLimit_MinX) OR
        ("DB_Manual".SelectedAxis = 1 AND #Axis_Z.StatusBits.HomingDone
         AND #Axis_Z.ActualPosition <= "DB_MachineConfig".SoftLimit_MinZ) OR
        #bToolAxisBlocked;
    // In STATE_PNP_HALT: additionally block jog direction that would drive the axis
    // deeper into the PNP zone. Jog toward the active PNP zone is blocked; jog away
    // (escape direction) is passed through.
    IF #State = STATE_PNP_HALT THEN
        "DB_Manual".Jog_Plus  := "DB_Manual".Btn_JogPlus AND NOT #bJogBlockPlus AND NOT (
            ("DB_Manual".SelectedAxis = 0 AND #HW_PNP_X_Max) OR
            ("DB_Manual".SelectedAxis = 1 AND #HW_PNP_Z_Max));
        "DB_Manual".Jog_Minus := "DB_Manual".Btn_JogMinus AND NOT #bJogBlockMinus AND NOT (
            ("DB_Manual".SelectedAxis = 0 AND #HW_PNP_X_Min) OR
            ("DB_Manual".SelectedAxis = 1 AND #HW_PNP_Z_Min));
    ELSE
        "DB_Manual".Jog_Plus  := "DB_Manual".Btn_JogPlus  AND NOT #bJogBlockPlus;
        "DB_Manual".Jog_Minus := "DB_Manual".Btn_JogMinus AND NOT #bJogBlockMinus;
    END_IF;
    // The interlock covers every manual command that can turn the turret, not just the
    // jog buttons: a MoveAbsolute or a Home on the tool axis breaks the pin exactly as
    // well as a jog does. HomeAll is gated on the lock alone, whatever axis is selected,
    // because its step 3 homes the tool.
    "DB_Manual".Btn_HomeAxis := "DB_Manual".Btn_Home AND NOT #bToolAxisBlocked;

    // ITEM-56d (2026-08-16): refuse BLIND COORDINATE moves while halted in the PNP zone.
    // The jog gate above blocks the direction that would drive deeper in, but MoveAbsolute,
    // GoSafe and GoZero were passed through ungated -- they drive to a fixed coordinate with no
    // knowledge of which sensor tripped, so from PNP_HALT the operator could send the axis
    // straight back into the zone the machine had just halted for. GoZero is the clearest case:
    // it targets 0,0, i.e. toward MIN, which is exactly the wrong way after a MIN trip.
    //
    // Home and HomeAll are DELIBERATELY NOT blocked. Homing is the escape, not a hazard -- it is
    // the same action the Reset -> Start recovery performs, FB_ManualMode states 40/50 already
    // pre-clear the min proximity zone before seeking (bClearX/Z := PNP_X/Z_Min), and the TO is
    // configured to reverse at the hardware limit. Blocking them would remove the operator's
    // manual way out and leave only the automatic one. An earlier draft of this item lumped all
    // five buttons together; that was wrong. The distinction is blind coordinate move vs
    // reference-seeking move -- keep it that way if this is ever revisited.
    #bBlindMoveBlocked := (#State = STATE_PNP_HALT);

    #fbManualMode(Enable := (#State = STATE_MANUAL OR #State = STATE_PNP_HALT),
                  SelectedAxis := "DB_Manual".SelectedAxis,
                  Jog_Plus := "DB_Manual".Jog_Plus, Jog_Minus := "DB_Manual".Jog_Minus,
                  JogSpeed := "DB_Manual".JogSpeed,
                  MoveAbsolute := "DB_Manual".Btn_MoveAbsolute AND NOT #bToolAxisBlocked
                                  AND NOT #bBlindMoveBlocked,
                  TargetPosition := "DB_Manual".MoveToPosition,
                  HomeAxis := "DB_Manual".Btn_HomeAxis,
                  HomeAll := "DB_Manual".Btn_HomeAll AND NOT #bToolLockEngaged,
                  HomingMode := "DB_Manual".HomingMode, HomePosition := 0.0,
                  GoSafe := "DB_Manual".Btn_GoSafe AND NOT #bBlindMoveBlocked,
                  GoZero := "DB_Manual".Btn_GoZero AND NOT #bBlindMoveBlocked,
                  SafeToJog := #fbSafetyMonitor.SafeToJog, Reset := #fbInputs.Cmd_Reset,
                  PNP_X_Min := #HW_PNP_X_Min, PNP_Z_Min := #HW_PNP_Z_Min,
                  // Turret-step buttons: the most direct way to rotate the turret from the
                  // panel, and they were the one hole left in the 2026-08-14 interlock.
                  // Gated on the lock alone -- see #bToolStepBlocked above.
                  ToolStepCW  := "DB_Manual".Btn_ToolStepCW  AND NOT #bToolLockEngaged,
                  ToolStepCCW := "DB_Manual".Btn_ToolStepCCW AND NOT #bToolLockEngaged,
                  ToolStepAngle := "DB_Manual".ToolStepAngle, ToolStepSpeed := "DB_Manual".ToolStepSpeed,
                  Axis_X := #Axis_X, Axis_Z := #Axis_Z, Axis_Tool := #Axis_Tool, Axis_Spindle := #Axis_Spindle);

    // Update manual mode status
    "DB_Manual".JogBusy := #fbManualMode.Busy;
    "DB_Manual".ManualBusy := #fbManualMode.Busy;       // Alias
    "DB_Manual".JogError := #fbManualMode.Error;
    "DB_Manual".ManualError := #fbManualMode.Error;     // Alias
    "DB_Manual".JogErrorID := #fbManualMode.ErrorID;
    "DB_Manual".ManualErrorID := #fbManualMode.ErrorID; // Alias
    "DB_Manual".SelectedAxisPos := SEL(G := "DB_Manual".SelectedAxis = 0,
                                        IN0 := #Axis_Z.ActualPosition, IN1 := #Axis_X.ActualPosition);
    "DB_Manual".SelectedAxisName := SEL(G := "DB_Manual".SelectedAxis = 0, IN0 := 'Z', IN1 := 'X');
    "DB_Manual".ToolPosition := #Axis_Tool.ActualPosition;
    "DB_Manual".ActiveAxis := #fbManualMode.ActiveAxis;

    // Forward manual mode errors to alarm manager (once, on rising edge)
    IF #fbManualMode.Error AND NOT #prevManualError THEN
        #newErrorFlag := TRUE;
        #newErrorCode := #fbManualMode.ErrorID;
        // Single-writer: ErrorText comes from the FB_AlarmManager CASE table for the code.
        // DB_HMI.ErrorDetail is written directly inside FB_ManualMode at each error point.
    END_IF;
    #prevManualError := #fbManualMode.Error;

    // =========================================================================
    // SPINDLE CONTROL
    // Manual mode spindle control via DB_Manual buttons
    // Recipe handler spindle control via bSpindleStart/bSpindleStop flags
    // =========================================================================
    // Capture inputs BEFORE calling the FB so Diag_* reflects this scan's values.
    "DB_Spindle".Diag_bSpindleStart := #bSpindleStart;
    "DB_Spindle".Diag_bSpindleStop  := #bSpindleStop;
    "DB_Spindle".Diag_EnableInput   := #bDrivesEnable;
    "DB_Spindle".Diag_StartInput    := "DB_Manual".Btn_SpindleStart OR #bSpindleStart;
    "DB_Spindle".Diag_StopInput     := "DB_Manual".Btn_SpindleStop OR #bSpindleStop OR #fbInputs.Cmd_Stop;
    "DB_Spindle".Diag_ReqStart      := #fbRecipeHandler.SpindleReqStart;
    "DB_Spindle".Diag_ReqStop       := #fbRecipeHandler.SpindleReqStop;
    // -------------------------------------------------------------------------
    // Spindle history ring buffer: push snapshot on any meaningful change.
    // Trigger fields: SpindleState, PrevStart, ReqStart, StartEdge.
    // Reading tip: sort Hist_Log[0..19] by .Seq to get chronological order.
    // -------------------------------------------------------------------------
    IF "DB_Spindle".Hist_Clear THEN
        "DB_Spindle".Hist_Head   := 0;
        "DB_Spindle".Hist_Count  := 0;
        "DB_Spindle".Hist_SeqNum := 0;
        "DB_Spindle".Hist_Clear  := FALSE;
    ELSIF ("DB_Spindle".Diag_SpindleState <> #prevSnap_State)
       OR ("DB_Spindle".Diag_PrevStart    <> #prevSnap_PrevStart)
       OR ("DB_Spindle".Diag_ReqStart     <> #prevSnap_ReqStart)
       OR ("DB_Spindle".Diag_StartEdge    <> #prevSnap_StartEdge)
       OR ("DB_Spindle".Diag_MoveVelBusy  <> #prevSnap_MoveVelBusy) THEN
        // Push new entry at Hist_Head
        "DB_Spindle".Hist_Log["DB_Spindle".Hist_Head].Seq          := "DB_Spindle".Hist_SeqNum;
        "DB_Spindle".Hist_Log["DB_Spindle".Hist_Head].MachineState := #State;
        "DB_Spindle".Hist_Log["DB_Spindle".Hist_Head].State        := "DB_Spindle".Diag_SpindleState;
        "DB_Spindle".Hist_Log["DB_Spindle".Hist_Head].ReqStart     := "DB_Spindle".Diag_ReqStart;
        "DB_Spindle".Hist_Log["DB_Spindle".Hist_Head].ReqStop      := "DB_Spindle".Diag_ReqStop;
        "DB_Spindle".Hist_Log["DB_Spindle".Hist_Head].bStart       := "DB_Spindle".Diag_bSpindleStart;
        "DB_Spindle".Hist_Log["DB_Spindle".Hist_Head].bStop        := "DB_Spindle".Diag_bSpindleStop;
        "DB_Spindle".Hist_Log["DB_Spindle".Hist_Head].StartInput   := "DB_Spindle".Diag_StartInput;
        "DB_Spindle".Hist_Log["DB_Spindle".Hist_Head].StopInput    := "DB_Spindle".Diag_StopInput;
        "DB_Spindle".Hist_Log["DB_Spindle".Hist_Head].EnableIn     := "DB_Spindle".Diag_EnableInput;
        "DB_Spindle".Hist_Log["DB_Spindle".Hist_Head].PrevStart    := "DB_Spindle".Diag_PrevStart;
        "DB_Spindle".Hist_Log["DB_Spindle".Hist_Head].StartEdge    := "DB_Spindle".Diag_StartEdge;
        "DB_Spindle".Hist_Log["DB_Spindle".Hist_Head].MoveVelBusy  := "DB_Spindle".Diag_MoveVelBusy;
        "DB_Spindle".Hist_Log["DB_Spindle".Hist_Head].MoveVelInVel := "DB_Spindle".Diag_MoveVelInVel;
        // Advance ring buffer pointer
        "DB_Spindle".Hist_SeqNum := "DB_Spindle".Hist_SeqNum + 1;
        "DB_Spindle".Hist_Head   := ("DB_Spindle".Hist_Head + 1) MOD 20;
        IF "DB_Spindle".Hist_Count < 20 THEN
            "DB_Spindle".Hist_Count := "DB_Spindle".Hist_Count + 1;
        END_IF;
        // Latch current values for next-scan comparison
        #prevSnap_State       := "DB_Spindle".Diag_SpindleState;
        #prevSnap_PrevStart   := "DB_Spindle".Diag_PrevStart;
        #prevSnap_ReqStart    := "DB_Spindle".Diag_ReqStart;
        #prevSnap_StartEdge   := "DB_Spindle".Diag_StartEdge;
        #prevSnap_MoveVelBusy := "DB_Spindle".Diag_MoveVelBusy;
    END_IF;
    // RunCmd is a level signal (TRUE = run).
    // The CALLER must:
    //   • Set SetSpeed before raising RunCmd
    //   • Lower RunCmd to stop (do not change SetSpeed while RunCmd is TRUE)
    //   • For a speed change: lower RunCmd → update SetSpeed → raise RunCmd again
    #fbSpindleControl(
        Enable   := #bDrivesEnable,
        // Spindle stops while paused (State=PAUSED and NOT yet in the resume spin-up
        // window). This drops RunForward only — no MC_Halt — so the PTO keeps pulsing
        // (VFD-safe stop, same mechanism as a normal stop). On Continue, bResumeSpeedup
        // re-enables it for the spin-up wait before the axes return.
        RunCmd   := ("DB_Manual".Btn_SpindleStart OR #bSpindleStart)
                    AND NOT ("DB_Manual".Btn_SpindleStop OR #bSpindleStop OR #fbInputs.Cmd_Stop
                             OR (#State = STATE_PAUSED AND NOT #bResumeSpeedup)),
        SetSpeed := SEL(G := (#State = STATE_MANUAL),
                        IN0 := "DB_Spindle".Cmd_SetSpeed,
                        IN1 := "DB_Manual".Manual_SpindleSpeed),
        SpeedOverride := "DB_Spindle".SpeedOverride,
        Reset    := #fbInputs.Cmd_Reset,
        AckError := #ackEdge OR "DB_Manual".Btn_SpindleAckError,
	RunForward := "PTO_RunForward_AxisS",
        Axis_Spindle := #Axis_Spindle
    );
    // Write FB outputs back to DB_Spindle so HMI tags reflect actual state
    "DB_Spindle".IsRunning    := #fbSpindleControl.Running;
    "DB_Spindle".AtSpeed      := #fbSpindleControl.AtSpeed;
    "DB_Spindle".ActualSpeed  := #fbSpindleControl.ActualSpeed;

    // =========================================================================
    // TOOLHEADLOCK CONTROL
    // Written every scan so FB_CylinderControl (called from OB1) sees the
    // correct command on the next scan.
    //
    // EXTEND (Sol_A ON):  STATE_RUNNING (20), STATE_PAUSED (25), STATE_LOCK_EXTEND_WAIT (17)
    // RETRACT (spring):   all other states -- cylinder retracts automatically via spring return.
    //
    // Safety: spring-return valve retracts on power loss without any PLC action.
    // State 17 checks AtSetpoint for extend confirmation only -- no fallback timer in FB_Process.
    // CylFB Timeout_Extend (T#6S in DB_Cylinder_ToolHeadLock) is the sole timer; on timeout
    // CylFB sets Error=TRUE, state 17 catches it and goes to STATE_ERROR (16#0012).
    // State 29 uses tonLockWait only (spring retract; no retract sensor).
    // =========================================================================
    "DB_Cylinder_ToolHeadLock".Cmd_Extend :=
        (#State = STATE_RUNNING) OR
        (#State = STATE_PAUSED) OR
        (#State = STATE_LOCK_EXTEND_WAIT AND #tonLockPreDelay.Q);

    // Diagnostic output
    "DB_Diagnostic".Process_State        := #State;
    "DB_Diagnostic".Process_SafeToRun    := #SafeToRun;
    "DB_Diagnostic".Process_DrivesEnable := #bDrivesEnable;
    "DB_Diagnostic".Recipe_CurrentProgram := #activeProgram;
    "DB_Diagnostic".Recipe_TotalLines    := #activeLineCount;
    "DB_Diagnostic".Axis_X_Pos           := #Axis_X.ActualPosition;
    "DB_Diagnostic".Axis_Z_Pos           := #Axis_Z.ActualPosition;
    "DB_Diagnostic".Axis_X_Enabled       := #fbPowerX.Status;
    "DB_Diagnostic".Axis_Z_Enabled       := #fbPowerZ.Status;
    "DB_Diagnostic".Axis_X_Homed         := #Axis_X.StatusBits.HomingDone;
    "DB_Diagnostic".Axis_Z_Homed         := #Axis_Z.StatusBits.HomingDone;

    // Loaded recipe name -> HMI (2026-08-10). CAM writes Header.sName; until now nothing
    // surfaced it, so the operator had no way to see WHICH program is about to run -- only
    // its slot number. That gets worse with 50 slots.
    //
    // A CONTINUOUS MIRROR, deliberately not a latched copy. It always reports the buffer's
    // real content, which is why it needs no entry in any of the four reset paths: there is
    // nothing to clear. It also inherits the loader's poison for free -- ST_LATCH sets
    // Header.sName := '' before the transfer starts, so a failed or in-flight load shows a
    // BLANK name rather than the previous program's, and a blank name next to a non-zero
    // slot number means "not loaded", never "loaded something else".
    //
    // Pair it with DB_Diagnostic.Recipe_LoadedProgram on the HMI: slot number + name +
    // loaded-slot is enough for an operator to catch a wrong selection before pressing Start.
    "DB_HMI".LoadedProgramName           := "DB_SelectedRecipe".Header.sName;
    // Sanding dwell in progress (2026-08-29). Continuous mirror of the FB_Process latch,
    // so it appears in no reset path by design -- it follows #bSandActive to FALSE on
    // every exit (dwell expiry, Start, Stop, hard reset, error).
    "DB_HMI".SandActive                  := #bSandActive;

    // Checksum pair, for the HMI (2026-08-14). Same continuous-mirror discipline as
    // the name above: written every scan, in no reset path, always reporting what is
    // actually in the buffer.
    //
    // WHY BOTH NUMBERS AND NOT JUST A MATCH FLAG: on a 16#0316 the question is not
    // "did it match" -- the error already says it did not. It is WHICH SIDE IS WRONG.
    // Three implementations of this algorithm exist (SpinningCam's, tools/
    // split_recipe_db.py, and FB_RecipeLoader). The first two are cross-verified
    // against each other; the SCL one is not verified against anything. So if these
    // two numbers disagree, the operator can read both off the screen and say which,
    // instead of assuming the recipe is bad and re-exporting a perfectly good file.
    // A single boolean would hide exactly the information needed.
    "DB_HMI".Checksum_Recipe             := "DB_SelectedRecipe".Header.Checksum;
    "DB_HMI".Checksum_Calculated         := #fbRecipeLoader.ChecksumCalc;
    "DB_HMI".Checksum_Verified           := #fbRecipeLoader.ChecksumOK;

    // Pass display (2026-09-06). "Line 47 of 99" tells an operator nothing -- the job is
    // described in passes, and the recipe header already reads "Op1: ROUGHING, 10 paso".
    // Fed by the CMD=50/51 marker lines SpinningCam emits when its PLC-mode option is on.
    //
    // Same continuous-mirror discipline as the name and checksum above, and for the same
    // reason: it is written every scan, appears in NO reset path, and always reports what
    // FB_RecipeHandler actually holds. The handler's own Reset block zeroes all four, so a
    // stop or a hard reset blanks the HMI without four more clears to keep in sync here.
    //
    // 0 means NO PASS INFORMATION -- and it means that in every case: the recipe carries no
    // markers (the CAM option was off), or execution has not reached the first marker yet.
    // Because there is only one meaning, the HMI needs only one rule: blank the group on 0.
    // Do NOT mirror these inside STATE_RUNNING next to DB_HMI.CurrentLine -- that would
    // freeze the last pass on screen after the program ends instead of clearing it.
    "DB_HMI".CurrentOp                   := #fbRecipeHandler.CurrentOp;
    "DB_HMI".TotalOps                    := #fbRecipeHandler.TotalOps;
    "DB_HMI".CurrentPass                 := #fbRecipeHandler.CurrentPass;
    "DB_HMI".TotalPasses                 := #fbRecipeHandler.TotalPasses;

    // =========================================================================
    // CONTACTOR CONTROL -- called as the last step of FB_Process.
    // FC_ContactorControl reads DB_HMI.Btn_Contactor_* and Bypass_EStop/HasError.
    // In auto mode STATE_STARTING already sets these flags TRUE; they are reflected to I/O here.
    // Called here rather than from OB1 to ensure contactor logic runs in sync with the process.
    // =========================================================================
    "FC_ContactorControl"();
END_FUNCTION_BLOCK
